// TIA Portal V17 export
// export: Created 2025-06-26T07:49:16.0857786Z, ExportSetting WithDefaults, DisplayName Totally Integrated Automation Portal, DisplayVersion V17 Update 8, DisplayName TIA Portal Openness, DisplayVersion V17 Update 8, DisplayName TIA Portal Version Control Interface, DisplayVersion V17, DisplayName STEP 7 Professional, DisplayVersion V17 Update 8, DisplayName STEP 7 Safety, DisplayVersion V17 Update 6, DisplayName WinCC Advanced, DisplayVersion V17 Update 8
ORGANIZATION_BLOCK "ModbusRTU"   // OB32, FBD, CyclicInterrupt
TITLE = Modbus RTU Communication
{ S7_Optimized_Access := 'TRUE' }
VERSION : 0.1
// Run the Modbus Master and place the fieldbus images into I/O memory
// stored: AutoNumber true, IsIECCheckEnabled false, SetENOAutomatically false
   VAR_INPUT
      Initial_Call : Bool;   // Initial call of this OB
      Event_Count : Int;   // Events discarded
   END_VAR
BEGIN

REGION Network 1
   // To enable communication, set bStart to TRUE
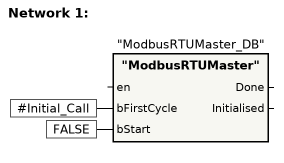
   "ModbusRTUMaster_DB"(bFirstCycle := #Initial_Call, bStart := FALSE);   // "ModbusRTUMaster"
END_REGION
END_ORGANIZATION_BLOCK
